SUBAPPLICATION Button_IXA_TO_logiBUS_QXA (* Konvertierung Button IXA zu logiBUS QXA *)
  (* Standard: 61499-2; Description: Copyright (c) 2023 Meisterschulen am Ostbahnhof This program and the accompanying materials are made available under the terms of the Eclipse Public License 2.0 which is available at https://www.eclipse.org/legal/epl-2.0/ SPDX-License-Identifier: EPL-2.0 *)
  (* Version 1.0, 2026-01-15, Franz Höpfinger, Meisterschulen am Ostbahnhof, initial API and implementation and/or initial documentation *)
  PACKAGE MyLib::sys;
  IMPORT isobus::UT::Q::const::IDs::ID_NULL;
  IMPORT logiBUS::io::DQ::logiBUS_DO;
  IMPORT logiBUS::io::DQ::logiBUS_DO_S;
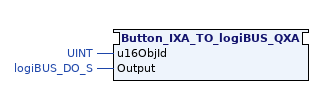
  VAR_INPUT
    u16ObjId : UINT := ID_NULL; (* Object ID *)
    Output : logiBUS::io::DQ::logiBUS_DO_S := logiBUS_DO::Invalid; (* Identify the Output Output_Q1..Q8 *)
  END_VAR
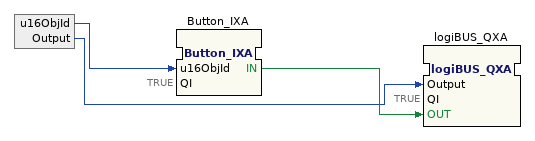
  FBS
    logiBUS_QXA : logiBUS::io::DQ::logiBUS_QXA(QI := TRUE);
    Button_IXA : isobus::UT::io::Button::Button_IXA(QI := TRUE);
  END_FBS
  DATA_CONNECTIONS
    u16ObjId TO Button_IXA.u16ObjId;
    Output TO logiBUS_QXA.Output;
  END_CONNECTIONS
  ADAPTER_CONNECTIONS
    Button_IXA.IN TO logiBUS_QXA.OUT;
  END_CONNECTIONS
END_SUBAPPLICATION
